// TIA Portal V16 export
// export: Created 2021-11-12T13:31:56.0731266Z, ExportSetting WithDefaults, DisplayName Totally Integrated Automation Portal, DisplayVersion V16 Update 3, DisplayName TIA Portal Version Control Interface, DisplayVersion V16 Update 2, DisplayName TIA Portal Openness, DisplayVersion V16 Update 3, DisplayName SINAMICS Startdrive Advanced, DisplayVersion V16 Update 5, DisplayName SINAMICS Startdrive G130, G150, S120, S150, SINAMICS MV, S210, DisplayVersion V16 Update 5, DisplayName SINAMICS Startdrive G110M, G120, G120C, G120D, G120P, G115D, DisplayVersion V16 Update 5, DisplayName STEP 7 Professional, DisplayVersion V16 Update 3, DisplayName STEP 7 Safety, DisplayVersion V16, DisplayName WinCC UA Professional, DisplayVersion V16 Update 3
FUNCTION_BLOCK "IM_000+UC20-KF10"   // FB49, LAD
TITLE = Inputs reading
{ S7_Optimized_Access := 'TRUE' }
VERSION : 0.1
// MICE Wood interface block
// stored: AutoNumber true, IsIECCheckEnabled false, IsRetainMemResEnabled false, MemoryReserve 100, SetENOAutomatically false, UDAEnableTagReadback false
   VAR
      KF11_Ix0 { S7_SetPoint := 'True'} : "STD_CH_DI";
      KF11_Ix1 { S7_SetPoint := 'True'} : "STD_CH_DI";
      KF11_Ix2 { S7_SetPoint := 'True'} : "STD_CH_DI";
      KF11_Ix3 { S7_SetPoint := 'True'} : "STD_CH_DI";
      KF11_Ix4 { S7_SetPoint := 'True'} : "STD_CH_DI";
      KF11_Ix5 { S7_SetPoint := 'True'} : "STD_CH_DI";
      KF11_Ix6 { S7_SetPoint := 'True'} : "STD_CH_DI";
      KF11_Ix7 { S7_SetPoint := 'True'} : "STD_CH_DI";
      KF12_Ix0 { S7_SetPoint := 'True'} : "STD_CH_DI";
      KF12_Ix1 { S7_SetPoint := 'True'} : "STD_CH_DI";
      KF12_Ix2 { S7_SetPoint := 'True'} : "STD_CH_DI";
      KF12_Ix3 { S7_SetPoint := 'True'} : "STD_CH_DI";
      KF12_Ix4 { S7_SetPoint := 'True'} : "STD_CH_DI";
      KF12_Ix5 { S7_SetPoint := 'True'} : "STD_CH_DI";
      KF12_Ix6 { S7_SetPoint := 'True'} : "STD_CH_DI";
      KF12_Ix7 { S7_SetPoint := 'True'} : "STD_CH_DI";
      KF13_Ix0 { S7_SetPoint := 'True'} : "STD_CH_DI";
      KF13_Ix1 { S7_SetPoint := 'True'} : "STD_CH_DI";
      KF13_Ix2 { S7_SetPoint := 'True'} : "STD_CH_DI";
      KF13_Ix3 { S7_SetPoint := 'True'} : "STD_CH_DI";
      KF13_Ix4 { S7_SetPoint := 'True'} : "STD_CH_DI";
      KF13_Ix5 { S7_SetPoint := 'True'} : "STD_CH_DI";
      KF13_Ix6 { S7_SetPoint := 'True'} : "STD_CH_DI";
      KF13_Ix7 { S7_SetPoint := 'True'} : "STD_CH_DI";
      KF14_Ix0 { S7_SetPoint := 'True'} : "STD_CH_DI";
      KF14_Ix1 { S7_SetPoint := 'True'} : "STD_CH_DI";
      KF14_Ix2 { S7_SetPoint := 'True'} : "STD_CH_DI";
      KF14_Ix3 { S7_SetPoint := 'True'} : "STD_CH_DI";
      KF14_Ix4 { S7_SetPoint := 'True'} : "STD_CH_DI";
      KF14_Ix5 { S7_SetPoint := 'True'} : "STD_CH_DI";
      KF14_Ix6 { S7_SetPoint := 'True'} : "STD_CH_DI";
      KF14_Ix7 { S7_SetPoint := 'True'} : "STD_CH_DI";
      KF15_Ix0 { S7_SetPoint := 'True'} : "STD_CH_DI";
      KF15_Ix1 { S7_SetPoint := 'True'} : "STD_CH_DI";
      KF15_Ix2 { S7_SetPoint := 'True'} : "STD_CH_DI";
      KF15_Ix3 { S7_SetPoint := 'True'} : "STD_CH_DI";
      KF15_Ix4 { S7_SetPoint := 'True'} : "STD_CH_DI";
      KF15_Ix5 { S7_SetPoint := 'True'} : "STD_CH_DI";
      KF15_Ix6 { S7_SetPoint := 'True'} : "STD_CH_DI";
      KF15_Ix7 { S7_SetPoint := 'True'} : "STD_CH_DI";
   END_VAR
   VAR_TEMP   // added for the SCL form of the ladder/FBD networks
      _w1 : Bool;
      _w2 : Bool;
      _w3 : Bool;
      _w4 : Bool;
   END_VAR
BEGIN

REGION Network 1: Module position -KF11
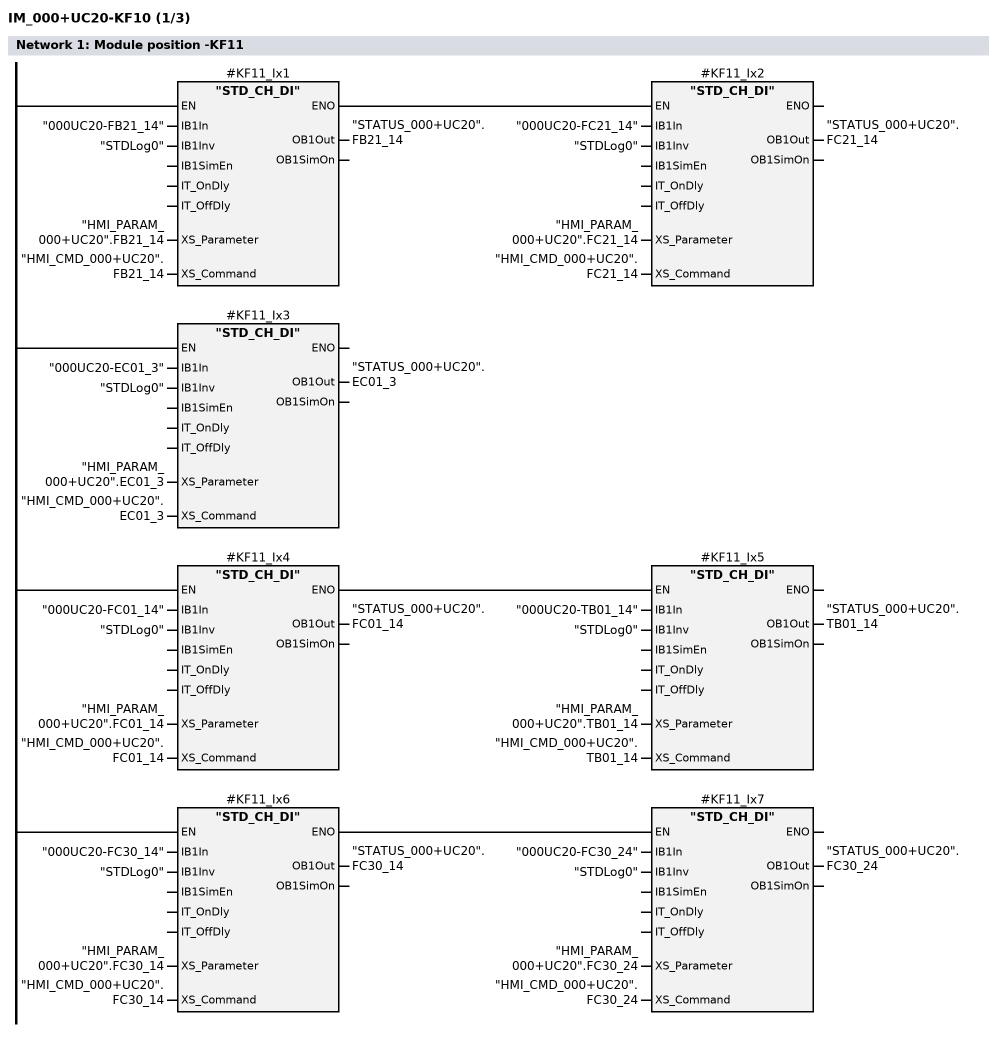
   RUNG wire#powerrail
      #KF11_Ix1(IB1In := "000UC20-FB21_14", IB1Inv := "STDLog0", IB1SimEn :=, IT_OnDly :=, IT_OffDly :=, XS_Parameter := "HMI_PARAM_000+UC20".FB21_14, XS_Command := "HMI_CMD_000+UC20".FB21_14, OB1Out => "STATUS_000+UC20".FB21_14, OB1SimOn =>)
      #KF11_Ix2(IB1In := "000UC20-FC21_14", IB1Inv := "STDLog0", IB1SimEn :=, IT_OnDly :=, IT_OffDly :=, XS_Parameter := "HMI_PARAM_000+UC20".FC21_14, XS_Command := "HMI_CMD_000+UC20".FC21_14, OB1Out => "STATUS_000+UC20".FC21_14, OB1SimOn =>)
   END_RUNG
   RUNG wire#powerrail
      #KF11_Ix3(IB1In := "000UC20-EC01_3", IB1Inv := "STDLog0", IB1SimEn :=, IT_OnDly :=, IT_OffDly :=, XS_Parameter := "HMI_PARAM_000+UC20".EC01_3, XS_Command := "HMI_CMD_000+UC20".EC01_3, OB1Out => "STATUS_000+UC20".EC01_3, OB1SimOn =>)
   END_RUNG
   RUNG wire#powerrail
      #KF11_Ix4(IB1In := "000UC20-FC01_14", IB1Inv := "STDLog0", IB1SimEn :=, IT_OnDly :=, IT_OffDly :=, XS_Parameter := "HMI_PARAM_000+UC20".FC01_14, XS_Command := "HMI_CMD_000+UC20".FC01_14, OB1Out => "STATUS_000+UC20".FC01_14, OB1SimOn =>)
      #KF11_Ix5(IB1In := "000UC20-TB01_14", IB1Inv := "STDLog0", IB1SimEn :=, IT_OnDly :=, IT_OffDly :=, XS_Parameter := "HMI_PARAM_000+UC20".TB01_14, XS_Command := "HMI_CMD_000+UC20".TB01_14, OB1Out => "STATUS_000+UC20".TB01_14, OB1SimOn =>)
   END_RUNG
   RUNG wire#powerrail
      #KF11_Ix6(IB1In := "000UC20-FC30_14", IB1Inv := "STDLog0", IB1SimEn :=, IT_OnDly :=, IT_OffDly :=, XS_Parameter := "HMI_PARAM_000+UC20".FC30_14, XS_Command := "HMI_CMD_000+UC20".FC30_14, OB1Out => "STATUS_000+UC20".FC30_14, OB1SimOn =>)
      #KF11_Ix7(IB1In := "000UC20-FC30_24", IB1Inv := "STDLog0", IB1SimEn :=, IT_OnDly :=, IT_OffDly :=, XS_Parameter := "HMI_PARAM_000+UC20".FC30_24, XS_Command := "HMI_CMD_000+UC20".FC30_24, OB1Out => "STATUS_000+UC20".FC30_24, OB1SimOn =>)
   END_RUNG
   // the same network as SCL:
   #KF11_Ix1(IB1In := "000UC20-FB21_14",   // "STD_CH_DI"
             IB1Inv := "STDLog0",
             XS_Parameter := "HMI_PARAM_000+UC20".FB21_14,
             XS_Command := "HMI_CMD_000+UC20".FB21_14,
             OB1Out => "STATUS_000+UC20".FB21_14,
             ENO => #_w1);
   IF #_w1 THEN
       #KF11_Ix2(IB1In := "000UC20-FC21_14",   // "STD_CH_DI"
                 IB1Inv := "STDLog0",
                 XS_Parameter := "HMI_PARAM_000+UC20".FC21_14,
                 XS_Command := "HMI_CMD_000+UC20".FC21_14,
                 OB1Out => "STATUS_000+UC20".FC21_14);
   END_IF;
   #KF11_Ix3(IB1In := "000UC20-EC01_3",   // "STD_CH_DI"
             IB1Inv := "STDLog0",
             XS_Parameter := "HMI_PARAM_000+UC20".EC01_3,
             XS_Command := "HMI_CMD_000+UC20".EC01_3,
             OB1Out => "STATUS_000+UC20".EC01_3);
   #KF11_Ix4(IB1In := "000UC20-FC01_14",   // "STD_CH_DI"
             IB1Inv := "STDLog0",
             XS_Parameter := "HMI_PARAM_000+UC20".FC01_14,
             XS_Command := "HMI_CMD_000+UC20".FC01_14,
             OB1Out => "STATUS_000+UC20".FC01_14,
             ENO => #_w2);
   IF #_w2 THEN
       #KF11_Ix5(IB1In := "000UC20-TB01_14",   // "STD_CH_DI"
                 IB1Inv := "STDLog0",
                 XS_Parameter := "HMI_PARAM_000+UC20".TB01_14,
                 XS_Command := "HMI_CMD_000+UC20".TB01_14,
                 OB1Out => "STATUS_000+UC20".TB01_14);
   END_IF;
   #KF11_Ix6(IB1In := "000UC20-FC30_14",   // "STD_CH_DI"
             IB1Inv := "STDLog0",
             XS_Parameter := "HMI_PARAM_000+UC20".FC30_14,
             XS_Command := "HMI_CMD_000+UC20".FC30_14,
             OB1Out => "STATUS_000+UC20".FC30_14,
             ENO => #_w3);
   IF #_w3 THEN
       #KF11_Ix7(IB1In := "000UC20-FC30_24",   // "STD_CH_DI"
                 IB1Inv := "STDLog0",
                 XS_Parameter := "HMI_PARAM_000+UC20".FC30_24,
                 XS_Command := "HMI_CMD_000+UC20".FC30_24,
                 OB1Out => "STATUS_000+UC20".FC30_24);
   END_IF;
END_REGION

REGION Network 2: Module position -KF12
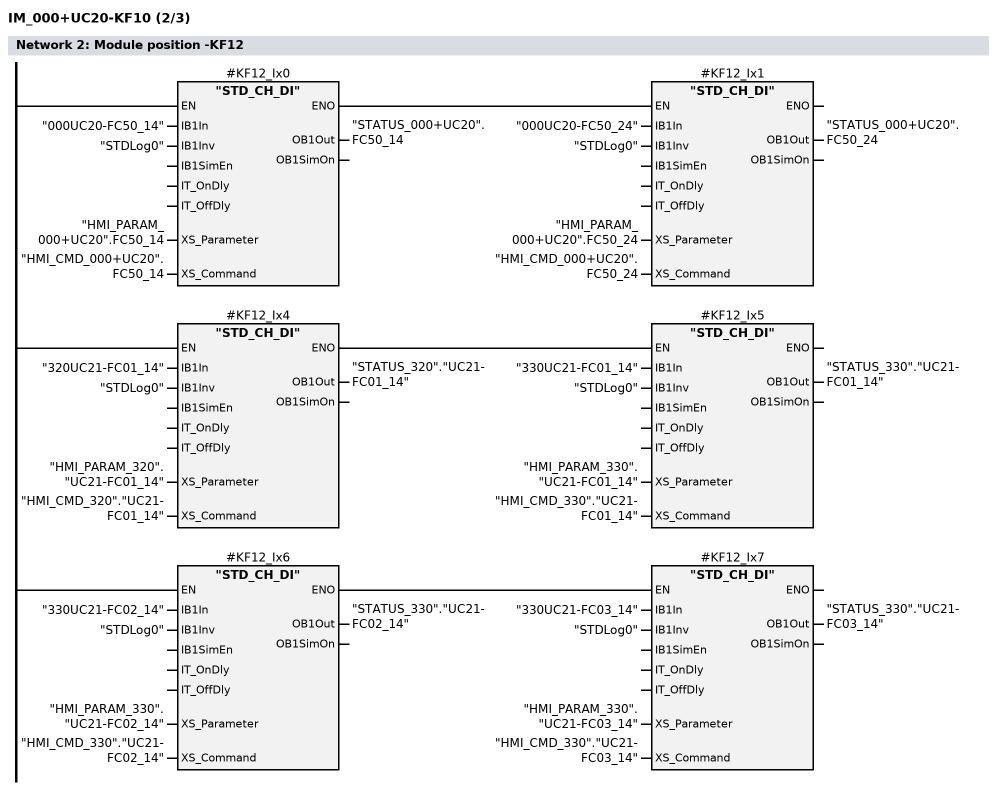
   RUNG wire#powerrail
      #KF12_Ix0(IB1In := "000UC20-FC50_14", IB1Inv := "STDLog0", IB1SimEn :=, IT_OnDly :=, IT_OffDly :=, XS_Parameter := "HMI_PARAM_000+UC20".FC50_14, XS_Command := "HMI_CMD_000+UC20".FC50_14, OB1Out => "STATUS_000+UC20".FC50_14, OB1SimOn =>)
      #KF12_Ix1(IB1In := "000UC20-FC50_24", IB1Inv := "STDLog0", IB1SimEn :=, IT_OnDly :=, IT_OffDly :=, XS_Parameter := "HMI_PARAM_000+UC20".FC50_24, XS_Command := "HMI_CMD_000+UC20".FC50_24, OB1Out => "STATUS_000+UC20".FC50_24, OB1SimOn =>)
   END_RUNG
   RUNG wire#powerrail
      #KF12_Ix4(IB1In := "320UC21-FC01_14", IB1Inv := "STDLog0", IB1SimEn :=, IT_OnDly :=, IT_OffDly :=, XS_Parameter := "HMI_PARAM_320"."UC21-FC01_14", XS_Command := "HMI_CMD_320"."UC21-FC01_14", OB1Out => "STATUS_320"."UC21-FC01_14", OB1SimOn =>)
      #KF12_Ix5(IB1In := "330UC21-FC01_14", IB1Inv := "STDLog0", IB1SimEn :=, IT_OnDly :=, IT_OffDly :=, XS_Parameter := "HMI_PARAM_330"."UC21-FC01_14", XS_Command := "HMI_CMD_330"."UC21-FC01_14", OB1Out => "STATUS_330"."UC21-FC01_14", OB1SimOn =>)
   END_RUNG
   RUNG wire#powerrail
      #KF12_Ix6(IB1In := "330UC21-FC02_14", IB1Inv := "STDLog0", IB1SimEn :=, IT_OnDly :=, IT_OffDly :=, XS_Parameter := "HMI_PARAM_330"."UC21-FC02_14", XS_Command := "HMI_CMD_330"."UC21-FC02_14", OB1Out => "STATUS_330"."UC21-FC02_14", OB1SimOn =>)
      #KF12_Ix7(IB1In := "330UC21-FC03_14", IB1Inv := "STDLog0", IB1SimEn :=, IT_OnDly :=, IT_OffDly :=, XS_Parameter := "HMI_PARAM_330"."UC21-FC03_14", XS_Command := "HMI_CMD_330"."UC21-FC03_14", OB1Out => "STATUS_330"."UC21-FC03_14", OB1SimOn =>)
   END_RUNG
   // the same network as SCL:
   #KF12_Ix0(IB1In := "000UC20-FC50_14",   // "STD_CH_DI"
             IB1Inv := "STDLog0",
             XS_Parameter := "HMI_PARAM_000+UC20".FC50_14,
             XS_Command := "HMI_CMD_000+UC20".FC50_14,
             OB1Out => "STATUS_000+UC20".FC50_14,
             ENO => #_w1);
   IF #_w1 THEN
       #KF12_Ix1(IB1In := "000UC20-FC50_24",   // "STD_CH_DI"
                 IB1Inv := "STDLog0",
                 XS_Parameter := "HMI_PARAM_000+UC20".FC50_24,
                 XS_Command := "HMI_CMD_000+UC20".FC50_24,
                 OB1Out => "STATUS_000+UC20".FC50_24);
   END_IF;
   #KF12_Ix4(IB1In := "320UC21-FC01_14",   // "STD_CH_DI"
             IB1Inv := "STDLog0",
             XS_Parameter := "HMI_PARAM_320"."UC21-FC01_14",
             XS_Command := "HMI_CMD_320"."UC21-FC01_14",
             OB1Out => "STATUS_320"."UC21-FC01_14",
             ENO => #_w2);
   IF #_w2 THEN
       #KF12_Ix5(IB1In := "330UC21-FC01_14",   // "STD_CH_DI"
                 IB1Inv := "STDLog0",
                 XS_Parameter := "HMI_PARAM_330"."UC21-FC01_14",
                 XS_Command := "HMI_CMD_330"."UC21-FC01_14",
                 OB1Out => "STATUS_330"."UC21-FC01_14");
   END_IF;
   #KF12_Ix6(IB1In := "330UC21-FC02_14",   // "STD_CH_DI"
             IB1Inv := "STDLog0",
             XS_Parameter := "HMI_PARAM_330"."UC21-FC02_14",
             XS_Command := "HMI_CMD_330"."UC21-FC02_14",
             OB1Out => "STATUS_330"."UC21-FC02_14",
             ENO => #_w3);
   IF #_w3 THEN
       #KF12_Ix7(IB1In := "330UC21-FC03_14",   // "STD_CH_DI"
                 IB1Inv := "STDLog0",
                 XS_Parameter := "HMI_PARAM_330"."UC21-FC03_14",
                 XS_Command := "HMI_CMD_330"."UC21-FC03_14",
                 OB1Out => "STATUS_330"."UC21-FC03_14");
   END_IF;
END_REGION

REGION Network 3: Module position -KF13
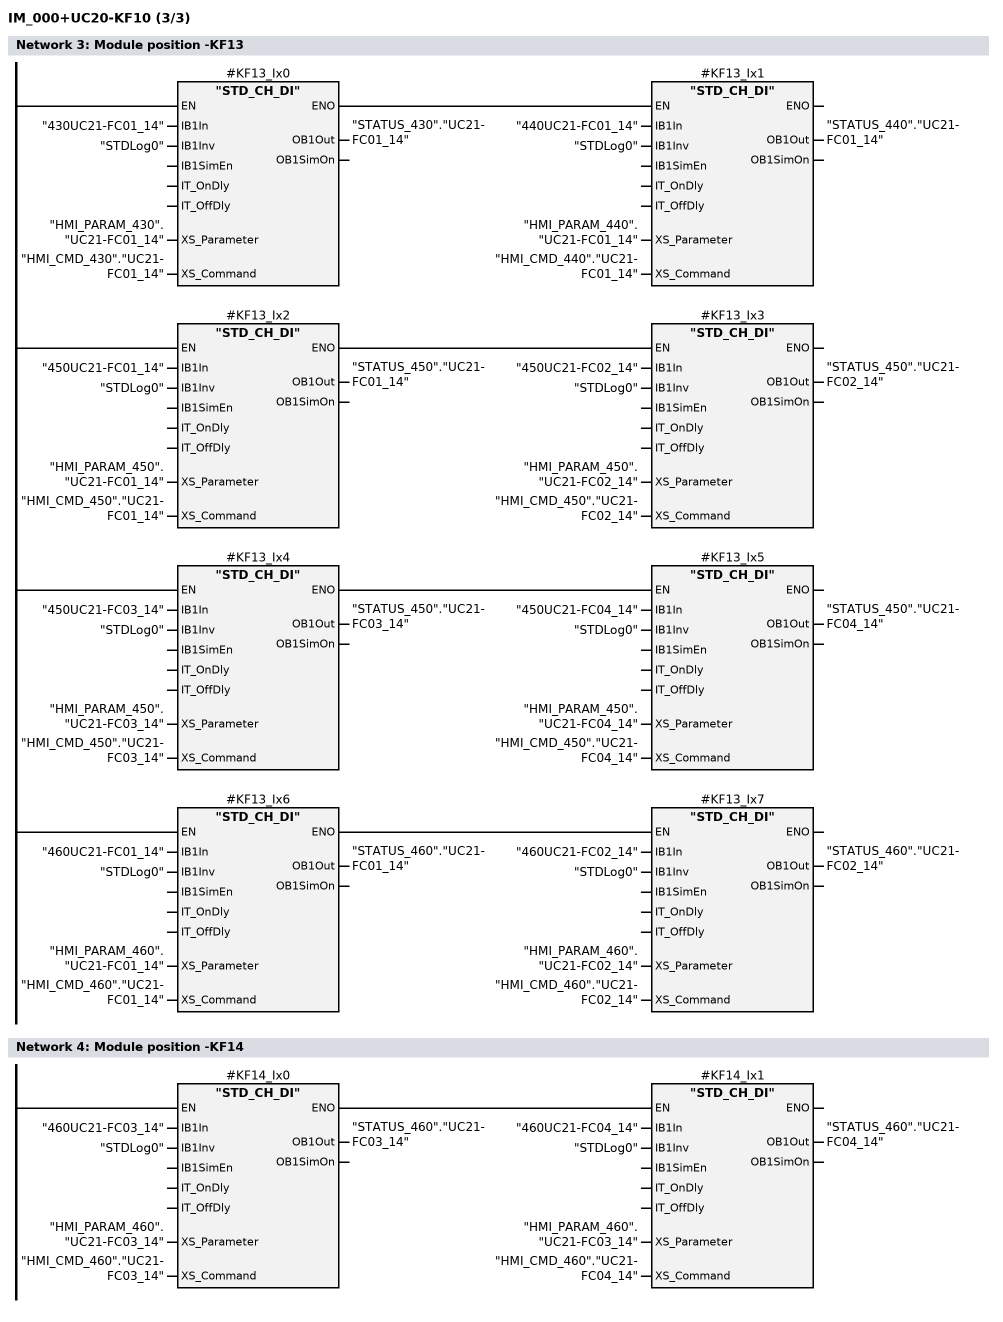
   RUNG wire#powerrail
      #KF13_Ix0(IB1In := "430UC21-FC01_14", IB1Inv := "STDLog0", IB1SimEn :=, IT_OnDly :=, IT_OffDly :=, XS_Parameter := "HMI_PARAM_430"."UC21-FC01_14", XS_Command := "HMI_CMD_430"."UC21-FC01_14", OB1Out => "STATUS_430"."UC21-FC01_14", OB1SimOn =>)
      #KF13_Ix1(IB1In := "440UC21-FC01_14", IB1Inv := "STDLog0", IB1SimEn :=, IT_OnDly :=, IT_OffDly :=, XS_Parameter := "HMI_PARAM_440"."UC21-FC01_14", XS_Command := "HMI_CMD_440"."UC21-FC01_14", OB1Out => "STATUS_440"."UC21-FC01_14", OB1SimOn =>)
   END_RUNG
   RUNG wire#powerrail
      #KF13_Ix2(IB1In := "450UC21-FC01_14", IB1Inv := "STDLog0", IB1SimEn :=, IT_OnDly :=, IT_OffDly :=, XS_Parameter := "HMI_PARAM_450"."UC21-FC01_14", XS_Command := "HMI_CMD_450"."UC21-FC01_14", OB1Out => "STATUS_450"."UC21-FC01_14", OB1SimOn =>)
      #KF13_Ix3(IB1In := "450UC21-FC02_14", IB1Inv := "STDLog0", IB1SimEn :=, IT_OnDly :=, IT_OffDly :=, XS_Parameter := "HMI_PARAM_450"."UC21-FC02_14", XS_Command := "HMI_CMD_450"."UC21-FC02_14", OB1Out => "STATUS_450"."UC21-FC02_14", OB1SimOn =>)
   END_RUNG
   RUNG wire#powerrail
      #KF13_Ix4(IB1In := "450UC21-FC03_14", IB1Inv := "STDLog0", IB1SimEn :=, IT_OnDly :=, IT_OffDly :=, XS_Parameter := "HMI_PARAM_450"."UC21-FC03_14", XS_Command := "HMI_CMD_450"."UC21-FC03_14", OB1Out => "STATUS_450"."UC21-FC03_14", OB1SimOn =>)
      #KF13_Ix5(IB1In := "450UC21-FC04_14", IB1Inv := "STDLog0", IB1SimEn :=, IT_OnDly :=, IT_OffDly :=, XS_Parameter := "HMI_PARAM_450"."UC21-FC04_14", XS_Command := "HMI_CMD_450"."UC21-FC04_14", OB1Out => "STATUS_450"."UC21-FC04_14", OB1SimOn =>)
   END_RUNG
   RUNG wire#powerrail
      #KF13_Ix6(IB1In := "460UC21-FC01_14", IB1Inv := "STDLog0", IB1SimEn :=, IT_OnDly :=, IT_OffDly :=, XS_Parameter := "HMI_PARAM_460"."UC21-FC01_14", XS_Command := "HMI_CMD_460"."UC21-FC01_14", OB1Out => "STATUS_460"."UC21-FC01_14", OB1SimOn =>)
      #KF13_Ix7(IB1In := "460UC21-FC02_14", IB1Inv := "STDLog0", IB1SimEn :=, IT_OnDly :=, IT_OffDly :=, XS_Parameter := "HMI_PARAM_460"."UC21-FC02_14", XS_Command := "HMI_CMD_460"."UC21-FC02_14", OB1Out => "STATUS_460"."UC21-FC02_14", OB1SimOn =>)
   END_RUNG
   // the same network as SCL:
   #KF13_Ix0(IB1In := "430UC21-FC01_14",   // "STD_CH_DI"
             IB1Inv := "STDLog0",
             XS_Parameter := "HMI_PARAM_430"."UC21-FC01_14",
             XS_Command := "HMI_CMD_430"."UC21-FC01_14",
             OB1Out => "STATUS_430"."UC21-FC01_14",
             ENO => #_w1);
   IF #_w1 THEN
       #KF13_Ix1(IB1In := "440UC21-FC01_14",   // "STD_CH_DI"
                 IB1Inv := "STDLog0",
                 XS_Parameter := "HMI_PARAM_440"."UC21-FC01_14",
                 XS_Command := "HMI_CMD_440"."UC21-FC01_14",
                 OB1Out => "STATUS_440"."UC21-FC01_14");
   END_IF;
   #KF13_Ix2(IB1In := "450UC21-FC01_14",   // "STD_CH_DI"
             IB1Inv := "STDLog0",
             XS_Parameter := "HMI_PARAM_450"."UC21-FC01_14",
             XS_Command := "HMI_CMD_450"."UC21-FC01_14",
             OB1Out => "STATUS_450"."UC21-FC01_14",
             ENO => #_w2);
   IF #_w2 THEN
       #KF13_Ix3(IB1In := "450UC21-FC02_14",   // "STD_CH_DI"
                 IB1Inv := "STDLog0",
                 XS_Parameter := "HMI_PARAM_450"."UC21-FC02_14",
                 XS_Command := "HMI_CMD_450"."UC21-FC02_14",
                 OB1Out => "STATUS_450"."UC21-FC02_14");
   END_IF;
   #KF13_Ix4(IB1In := "450UC21-FC03_14",   // "STD_CH_DI"
             IB1Inv := "STDLog0",
             XS_Parameter := "HMI_PARAM_450"."UC21-FC03_14",
             XS_Command := "HMI_CMD_450"."UC21-FC03_14",
             OB1Out => "STATUS_450"."UC21-FC03_14",
             ENO => #_w3);
   IF #_w3 THEN
       #KF13_Ix5(IB1In := "450UC21-FC04_14",   // "STD_CH_DI"
                 IB1Inv := "STDLog0",
                 XS_Parameter := "HMI_PARAM_450"."UC21-FC04_14",
                 XS_Command := "HMI_CMD_450"."UC21-FC04_14",
                 OB1Out => "STATUS_450"."UC21-FC04_14");
   END_IF;
   #KF13_Ix6(IB1In := "460UC21-FC01_14",   // "STD_CH_DI"
             IB1Inv := "STDLog0",
             XS_Parameter := "HMI_PARAM_460"."UC21-FC01_14",
             XS_Command := "HMI_CMD_460"."UC21-FC01_14",
             OB1Out => "STATUS_460"."UC21-FC01_14",
             ENO => #_w4);
   IF #_w4 THEN
       #KF13_Ix7(IB1In := "460UC21-FC02_14",   // "STD_CH_DI"
                 IB1Inv := "STDLog0",
                 XS_Parameter := "HMI_PARAM_460"."UC21-FC02_14",
                 XS_Command := "HMI_CMD_460"."UC21-FC02_14",
                 OB1Out => "STATUS_460"."UC21-FC02_14");
   END_IF;
END_REGION

REGION Network 4: Module position -KF14
   RUNG wire#powerrail
      #KF14_Ix0(IB1In := "460UC21-FC03_14", IB1Inv := "STDLog0", IB1SimEn :=, IT_OnDly :=, IT_OffDly :=, XS_Parameter := "HMI_PARAM_460"."UC21-FC03_14", XS_Command := "HMI_CMD_460"."UC21-FC03_14", OB1Out => "STATUS_460"."UC21-FC03_14", OB1SimOn =>)
      #KF14_Ix1(IB1In := "460UC21-FC04_14", IB1Inv := "STDLog0", IB1SimEn :=, IT_OnDly :=, IT_OffDly :=, XS_Parameter := "HMI_PARAM_460"."UC21-FC03_14", XS_Command := "HMI_CMD_460"."UC21-FC04_14", OB1Out => "STATUS_460"."UC21-FC04_14", OB1SimOn =>)
   END_RUNG
   // the same network as SCL:
   #KF14_Ix0(IB1In := "460UC21-FC03_14",   // "STD_CH_DI"
             IB1Inv := "STDLog0",
             XS_Parameter := "HMI_PARAM_460"."UC21-FC03_14",
             XS_Command := "HMI_CMD_460"."UC21-FC03_14",
             OB1Out => "STATUS_460"."UC21-FC03_14",
             ENO => #_w1);
   IF #_w1 THEN
       #KF14_Ix1(IB1In := "460UC21-FC04_14",   // "STD_CH_DI"
                 IB1Inv := "STDLog0",
                 XS_Parameter := "HMI_PARAM_460"."UC21-FC03_14",
                 XS_Command := "HMI_CMD_460"."UC21-FC04_14",
                 OB1Out => "STATUS_460"."UC21-FC04_14");
   END_IF;
END_REGION
END_FUNCTION_BLOCK
